FUNCTION_BLOCK differential_protection_2 (* Basic Function Block Type *)
  (* Standard: 61499-2 *)
  (* Version 0.0, 3/23/2016, gulzha, nxtControl GmbH, Template *)
  PACKAGE Main;
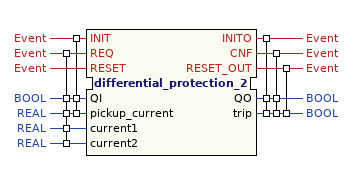
  EVENT_INPUT
    INIT WITH QI, pickup_current; (* Initialization Request *)
    REQ WITH QI, pickup_current, current1, current2; (* Normal Execution Request *)
    RESET;
  END_EVENT
  EVENT_OUTPUT
    INITO WITH QO, trip; (* Initialization Confirm *)
    CNF WITH QO, trip; (* Execution Confirmation *)
    RESET_OUT WITH trip;
  END_EVENT
  VAR_INPUT
    QI : BOOL; (* Input event qualifier *)
    pickup_current : REAL;
    current1 : REAL;
    current2 : REAL;
  END_VAR
  VAR_OUTPUT
    QO : BOOL; (* Output event qualifier *)
    trip : BOOL;
  END_VAR
  VAR
    fault : BOOL;
    differential : REAL;
    time2 : BOOL;
  END_VAR
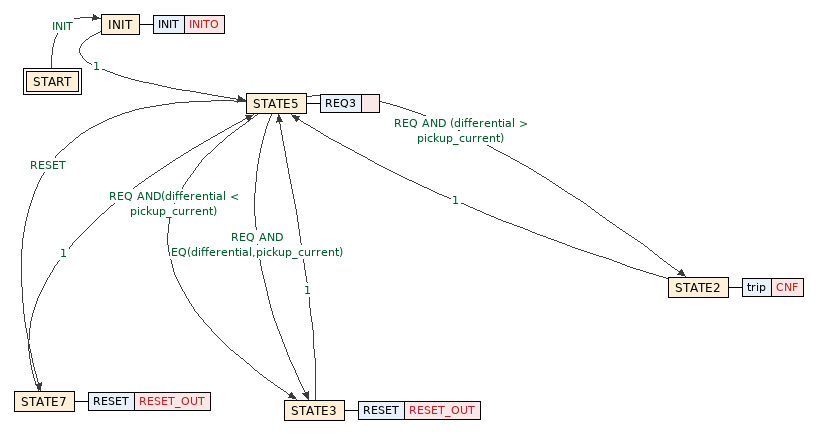
  EC_STATES
    START; (* Initial State *)
    INIT : INIT -> INITO; (* Initialization *)
    STATE2 : trip -> CNF;
    STATE3 : RESET -> RESET_OUT;
    STATE5 : REQ3;
    STATE7 : RESET -> RESET_OUT;
  END_STATES
  EC_TRANSITIONS
    START TO INIT := INIT;
    STATE5 TO STATE3 := REQ AND(differential < pickup_current);
    STATE7 TO STATE5 := 1;
    STATE5 TO STATE7 := RESET;
    STATE5 TO STATE2 := REQ AND (differential > pickup_current);
    INIT TO STATE5 := 1;
    STATE3 TO STATE5 := 1;
    STATE2 TO STATE5 := 1;
    STATE5 TO STATE3 := REQ AND EQ(differential,pickup_current);
  END_TRANSITIONS
  ALGORITHM INIT IN ST: (* Initialization algorithm *)
trip := FALSE;
fault := FALSE;
time2 := FALSE;

;
  END_ALGORITHM
  ALGORITHM trip IN ST: (* Normally executed algorithm *)
trip := TRUE;
;
  END_ALGORITHM
  ALGORITHM RESET IN ST:
trip := FALSE;
fault := FALSE;
time2 := FALSE;

;
  END_ALGORITHM
  ALGORITHM REQ2 IN ST:
fault := TRUE;
//REQ:=FALSE;
;
  END_ALGORITHM
  ALGORITHM REQ3 IN ST:
differential := ABS(current1 - current2);
//REQ := FALSE;
;
  END_ALGORITHM
  ALGORITHM time2_up IN ST:
time2 := TRUE;
;
  END_ALGORITHM
END_FUNCTION_BLOCK
